PROGRAM MAIN
VAR
	init_done		: BOOL := FALSE;
	
	//strategy controller
	Strategy : FB_BaseStrategyController; 

	//states thermal networks
	cnState : ST_BufferStorageState;
	hnltState : ST_BufferStorageState;
	hnhtState : ST_BufferStorageState;
	
	//thermal networks
	CN : FB_CoolingNetwork;
	HNLT_CN : FB_HnltCnLinkage;
	HNHT_CN : FB_HnhtCnLinkage;
	HNLT : FB_HeatingNetworkLowTemperature;
	HNHT_HNLT : FB_HnhtHnltLinkage;
	HNHT : FB_HeatingNetworkHighTemperature;
	
	//ambient state
	Ambient : FB_Ambient;
END_VAR

//implement states and linked them to exisiting buffer storage components
hnltState.fLowerTemperature := Speicher.Pufferspeicher_Warmwasser_295.Zustand.Temp_unten;
hnltState.fMidTemperature := Speicher.Pufferspeicher_Warmwasser_295.Zustand.Temp_mitte;
hnltState.fUpperTemperature := Speicher.Pufferspeicher_Warmwasser_295.Zustand.Temp_oben;
hnhtState.fUpperTemperature := Speicher.Pufferspeicher_Heisswasser_395.Zustand.Temp_oben;
hnhtState.fMidTemperature := Speicher.Pufferspeicher_Heisswasser_395.Zustand.Temp_mitte;
hnhtState.fLowerTemperature := Speicher.Pufferspeicher_Heisswasser_395.Zustand.Temp_unten;

//strategy controller
Strategy(ambientState := Ambient.localState,
	cnState := CN.localState,
	hnltState := hnltState,
	hnhtState := hnhtState);

//ambient state
Ambient();
	
//thermal networks
CN(controlAutomatic := Strategy.cnControl);

HNLT_CN(controlAutomatic := Strategy.hnltCnLinkageControl,
	stAmbientState := Ambient.localState);
	
HNHT_CN(controlAutomatic := Strategy.hnhtCnLinkageControl);
	
HNLT(ambientState := Ambient.localState,
	controlAutomatic := Strategy.hnltControl);
	
HNHT_HNLT(controlAutomatic := Strategy.hnhtHnltLinkageControl);
	
HNHT(controlAutomatic := Strategy.hnhtControl);

//Current implementation

(* --------------------------------------------------------------------------------------------------------------------------- *)

(* Analog- & Binaer Eingaenge - LESEN *)
(* P_Lesen; *)

	(* BUS Kommunikation - LESEN *)

(* --------------------------------------------------------------------------------------------------------------------------- *)
(* Starte Sub-Applikationen *)


	(*Initialisierung des Systems*)
	(*Einmalige Initialisierung der Parameter bei Hochlauf*)
	IF(NOT init_done) THEN
		Initialisierungsroutine();
		init_done := TRUE;
	END_IF;

	(* Allgemeine Parameter (Systemszeit, usw.) *)
	GA_Allgemein();

	(* Wandler *)
	Wandler();

	(* Speicher *)
	Speicher();

	(* Netze *)
	Netze();

	(* Management *)
	Management();

	(* Beleuchtung *)
	Beleuchtung();

	(*Anlagenversorgung*)
	Anlagenversorgung();

	(*Heizung Lüftung Klimatisierung*)
	Heizung_Lueftung_Klima();

	(*Umwelt*)
	Umwelt();

	(* Signal_Ampel *)
	Signal_Ampel();


	(*Test OPC-UA*)


	(*
	FAC_JAVA_READ_BOOL();
	MAFAC_JAVA_Read_REAL();
	IVA_Ofen_Read_BOOL();
	IVA_Ofen_Read_REAL();
*)
	(*PRG_Read_LREAL();*)



(* --------------------------------------------------------------------------------------------------------------------------- *)
(* Analog- & Binaer Ausgaenge - SCHREIBEN *)
(* P_Schreiben; *)

(* BUS Kommunikation - SCHREIBEN *)

END_PROGRAM

(* stored: Version 1.1.0.1, ProductVersion 3.1.4024.10
   POU MAIN: Id {f4373c39-f5a7-4799-b8f8-e268e2a0cb7c}, SpecialFunc None *)
